DATA_BLOCK "EM_Carriage_Drive_DB"
{ S7_Optimized_Access := 'TRUE' }
VERSION : 0.1
"EM_Carriage_Drive"
BEGIN
END_DATA_BLOCK
